// TwinCAT 3 PLC project Katas
// ProgramVersion: 3.1.4024.0
// libraries:
//   Tc2_Standard, * (Beckhoff Automation GmbH)
//   Tc2_System, * (Beckhoff Automation GmbH)
//   Tc3_Module, * (Beckhoff Automation GmbH)
// project tree:
//   / PlcTask.TcTTO
//   POUs/ MAIN.TcPOU, SevenSegmentDisplay.TcPOU
//   POUs/SortYourNumbers/ AscendingBubbleSort.TcPOU, SortYourNumbers.TcPOU
// real-time tasks:
//   TASK PlcTask: cycle T#10ms, priority 20, ADS port 350

CONFIGURATION Katas
    RESOURCE PLC ON TwinCAT3
        TASK PlcTask(INTERVAL := T#10ms, PRIORITY := 20);
        PROGRAM MAIN WITH PlcTask : MAIN;
    END_RESOURCE
END_CONFIGURATION

// ---- POUs/MAIN.TcPOU
PROGRAM MAIN
VAR
END_VAR

SortYourNumbers();
SevenSegmentDisplay();

END_PROGRAM

// ---- POUs/SortYourNumbers/SortYourNumbers.TcPOU
PROGRAM SortYourNumbers
VAR
	TestArray : ARRAY[0..9] OF INT := [1,3,8,5,2,9,4,7,6,10];
	SortFinished : BOOL;
	Loop: UINT;
	Temp: INT;
	SwapHappened: BOOL;
END_VAR

//WHILE NOT SortFinished DO
//	IF Loop < ((SIZEOF(TestArray)/2)-1) THEN
//		IF TestArray[Loop] > TestArray[Loop + 1] THEN
//			Temp := TestArray[Loop];
//			TestArray[Loop] := TestArray[Loop + 1];
//			TestArray[Loop + 1] := Temp;
//			SwapHappened := TRUE;
//		END_IF
//		Loop := Loop + 1;
//	ELSE
//		IF SwapHappened THEN
//			SwapHappened := FALSE;
//			Loop := 0;
//		ELSE
//			SortFinished := TRUE;
//		END_IF
//	END_IF
//END_WHILE

AscendingBubbleSort(ArrayToSort := TestArray);

END_PROGRAM

// ---- POUs/SortYourNumbers/AscendingBubbleSort.TcPOU
FUNCTION AscendingBubbleSort : BOOL
VAR_INPUT
END_VAR
VAR
	i: DINT;
	j: DINT;
	swap: INT;
	Swapped: BOOL;
END_VAR
VAR_IN_OUT
	ArrayToSort : array[*] of int;
END_VAR

FOR i := 0 TO UPPER_BOUND(ArrayToSort,1) DO
	Swapped := FALSE;
	FOR j := 0 TO (UPPER_BOUND(ArrayToSort,1) -1) DO
		IF ArrayToSort[j] > ArrayToSort[j+1] THEN
			swap := ArrayToSort[j];
			ArrayToSort[j] := ArrayToSort[j + 1];
			ArrayToSort[j+1] := swap;
			Swapped := TRUE;
		END_IF
	END_FOR
	IF NOT Swapped THEN
		EXIT;
	END_IF
END_FOR

END_FUNCTION

// ---- POUs/SevenSegmentDisplay.TcPOU
PROGRAM SevenSegmentDisplay
VAR
//					0
//				------
//			   1|	  | 5
//				---6---
//			   2|     | 4
//				------
//				   3
	SevenSegmentOut : ARRAY[0..6] OF BOOL;
	SevenSegmentConversion : BYTE;
	SevenSegmentDisplay : INT;
END_VAR

IF SevenSegmentDisplay >= 0 AND SevenSegmentDisplay <= 9 THEN
	CASE SevenSegmentDisplay OF
		0:
			SevenSegmentConversion := 126;
		1:
			SevenSegmentConversion := 6;
		2:
			SevenSegmentConversion := 91;
		3:
			SevenSegmentConversion := 79;
		4:
			SevenSegmentConversion := 39;
		5:
			SevenSegmentConversion := 109;
		6:
			SevenSegmentConversion := 125;
		7:
			SevenSegmentConversion := 70;
		8:
			SevenSegmentConversion := 127;
		9:
			SevenSegmentConversion := 103;
	END_CASE
	SevenSegmentOut[0] := SevenSegmentConversion.6;
	SevenSegmentOut[1] := SevenSegmentConversion.5;
	SevenSegmentOut[2] := SevenSegmentConversion.4;
	SevenSegmentOut[3] := SevenSegmentConversion.3;
	SevenSegmentOut[4] := SevenSegmentConversion.2;
	SevenSegmentOut[5] := SevenSegmentConversion.1;
	SevenSegmentOut[6] := SevenSegmentConversion.0;
END_IF

END_PROGRAM
